TYPE RFType :
(
	RFType_Default := 0 //常规分子泵
)UINT;
END_TYPE

(* stored: Version 1.1.0.1, ProductVersion 3.1.4024.4
   DUT RFType: Id {647c13cf-f53f-4996-9d75-9f371e1d9e19} *)
